FUNCTION_BLOCK ObserveRFC
VAR_INPUT
END_VAR
VAR_OUTPUT
END_VAR
VAR
	m_ptrRFC: POINTER TO RefeedingConveyor;
	m_ptrRFCWP1: POINTER TO xPPUProduct;
	m_ptrRFCWP2: POINTER TO xPPUProduct;
END_VAR

METHOD FB_init : BOOL
VAR_INPUT
	bInitRetains : BOOL; // if TRUE, the retain variables are initialized (warm start / cold start)
	bInCopyCode : BOOL;  // if TRUE, the instance afterwards gets moved into the copy code (online change)
	
	i_ptrRFC: POINTER TO RefeedingConveyor;
	i_ptrWP1: POINTER TO xPPUProduct;
	i_ptrWP2: POINTER TO xPPUProduct;
END_VAR
m_ptrRFC := i_ptrRFC;
m_ptrRFCWP1 := i_ptrWP1;
m_ptrRFCWP2 := i_ptrWP2;
END_METHOD

METHOD ResetDefinition : BOOL
VAR_INPUT
END_VAR
;
END_METHOD

(* Update an instance of ProcessState with the part of the process that can be observed by this Hardware Interface. *)
METHOD UpdateProcessObservation : BOOL
VAR_IN_OUT
	io_processState: ProcessState;
END_VAR
io_processState.UpdateState_Binary(EProcessVariables.RFC_WPAtStart, m_ptrRFC^.WPAtStart, TRUE);
io_processState.UpdateState_Binary(EProcessVariables.RFC_WPAtEnd, m_ptrRFC^.WPAtEnd, TRUE);
io_processState.UpdateState_Binary(EProcessVariables.RFC_SwitchExtended, m_ptrRFC^.m_Switch.Extended, TRUE);
io_processState.UpdateState_Binary(EProcessVariables.RFC_SwitchRetracted, m_ptrRFC^.m_Switch.Retracted, TRUE);

io_processState.UpdateState_Defined(EProcessVariables.RFC_WPAtStart, TRUE);
io_processState.UpdateState_Defined(EProcessVariables.RFC_WPAtEnd, TRUE);
io_processState.UpdateState_Defined(EProcessVariables.RFC_SwitchExtended, TRUE);
io_processState.UpdateState_Defined(EProcessVariables.RFC_SwitchRetracted, TRUE);
END_METHOD

END_FUNCTION_BLOCK

(* stored: Version 1.1.0.1
   POU ObserveRFC: Id {b84e58ee-1595-4bde-8682-8f02de2955d1}, SpecialFunc None
   Method FB_init: Id {bcc9372f-b1e5-4ed6-b565-314ff2f50d97}
   Method ResetDefinition: Id {1dea0e9f-7a7d-4c52-8f14-236af4a15989}
   Method UpdateProcessObservation: Id {93a85d47-e85b-45e4-893e-d6aa395d9f87} *)
